(* IEC 61131-3 sources: repolevel_ST_code_completion/output/0121完整版本/repoeval_three-axis_CNC_motion/readful_result_before_fix, 5 files *)

(* ---- INIT_CNC_System.st ---- *)
FUNCTION INIT_CNC_System : BOOL
VAR_IN_OUT
	fbSMC_ReadNCFile		:	SMC_ReadNCFile;
	fbSMC_NCDecoder			:	SMC_NCDecoder;
	fbSMC_CheckVelocities	:	SMC_CheckVelocities;
	fbSMC_Interpolator		:	SMC_Interpolator;
	fbSMC_ControlAxisXByPos	:	SMC_ControlAxisByPos;
	fbSMC_ControlAxisYByPos	:	SMC_ControlAxisByPos;
	fbSMC_ControlAxisZByPos	:	SMC_ControlAxisByPos;
	fbSMC_AXISX_HOMING		:	SMC_HOMING;
	fbSMC_AXISY_HOMING		:	SMC_HOMING;
	fbSMC_AXISZ_HOMING		:	SMC_HOMING;
	fbMC_AXISX_STOP			:	MC_STOP;
	fbMC_AXISY_STOP			:	MC_STOP;
	fbMC_AXISZ_STOP			:	MC_STOP;
END_VAR
VAR_INPUT
	AxisX					:	SM3_Basic.AXIS_REF_SM3
	AxisY					:	SM3_Basic.AXIS_REF_SM3
	AxisZ					:	SM3_Basic.AXIS_REF_SM3
END_VAR
VAR
	bInitSuccess : BOOL;
END_VAR

// Reset G-code processing related function blocks
fbSMC_ReadNCFile(bExecute := FALSE);
fbSMC_NCDecoder(bExecute := FALSE, ncprog := fbSMC_ReadNCFile.ncprog);
fbSMC_CheckVelocities(bExecute := FALSE);
fbSMC_Interpolator(bExecute := FALSE);

// Stop all axes
fbMC_AXISX_STOP(Axis := AxisX, Execute := TRUE);
fbMC_AXISY_STOP(Axis := AxisY, Execute := TRUE);
fbMC_AXISZ_STOP(Axis := AxisZ, Execute := TRUE);

// Perform homing for all axes
fbSMC_AXISX_HOMING(Axis := AxisX, Execute := TRUE);
fbSMC_AXISY_HOMING(Axis := AxisY, Execute := TRUE);
fbSMC_AXISZ_HOMING(Axis := AxisZ, Execute := TRUE);

// Check if initialization was successful
bInitSuccess := fbMC_AXISX_STOP.Done AND fbMC_AXISY_STOP.Done AND fbMC_AXISZ_STOP.Done AND
                fbSMC_AXISX_HOMING.Done AND fbSMC_AXISY_HOMING.Done AND fbSMC_AXISZ_HOMING.Done;

RETURN bInitSuccess;
END_FUNCTION

(* ---- FB_TripleAxisHoming.st ---- *)
FUNCTION_BLOCK FB_TripleAxisHoming
VAR_INPUT
	bExecute			:	BOOL;				//执行回零信号
	AxisX				:	AXIS_REF;			//X轴引用
	AxisY				:	AXIS_REF;			//Y轴引用
	AxisZ				:	AXIS_REF;			//Z轴引用
	bAxisXRefSwitch		:	BOOL;				//X轴零点开关
	bAxisYRefSwitch		:	BOOL;				//Y轴零点开关
	bAxisZRefSwitch		:	BOOL;				//Z轴零点开关
	fVelocitySlow		:	REAL;				//慢速回零速度
	fVelocityFast		:	REAL;				//快速回零速度
	fAcceleration		:	REAL;				//加速度
	fDeceleration		:	REAL;				//减速度
END_VAR
VAR_OUTPUT
	bHomeOK				:	BOOL;				//三轴都回零完成
	bAxisXHomeOK		:	BOOL;				//X轴回零完成
	bAxisYHomeOK		:	BOOL;				//Y轴回零完成
	bAxisZHomeOK		:	BOOL;				//Z轴回零完成
	bBusy				:	BOOL;				//回零进行中
	bError				:	BOOL;				//错误标志
	sErrorString		:	STRING;				//错误信息字符串
END_VAR
VAR
	fbHomingX			:	SMC_HOMING;			//X轴回零功能块
	fbHomingY			:	SMC_HOMING;			//Y轴回零功能块
	fbHomingZ			:	SMC_HOMING;			//Z轴回零功能块
	bAxisXBusy			:	BOOL;				//X轴回零进行中
	bAxisYBusy			:	BOOL;				//Y轴回零进行中
	bAxisZBusy			:	BOOL;				//Z轴回零进行中
	bAxisXError			:	BOOL;				//X轴回零错误
	bAxisYError			:	BOOL;				//Y轴回零错误
	bAxisZError			:	BOOL;				//Z轴回零错误
	sAxisXErrorString	:	STRING;				//X轴错误信息
	sAxisYErrorString	:	STRING;				//Y轴错误信息
	sAxisZErrorString	:	STRING;				//Z轴错误信息
END_VAR

fbHomingX.Execute := bExecute;
fbHomingX.Axis := AxisX;
fbHomingX.ReferenceSwitch := bAxisXRefSwitch;
fbHomingX.VelocitySlow := fVelocitySlow;
fbHomingX.VelocityFast := fVelocityFast;
fbHomingX.Acceleration := fAcceleration;
fbHomingX.Deceleration := fDeceleration;

fbHomingY.Execute := bExecute;
fbHomingY.Axis := AxisY;
fbHomingY.ReferenceSwitch := bAxisYRefSwitch;
fbHomingY.VelocitySlow := fVelocitySlow;
fbHomingY.VelocityFast := fVelocityFast;
fbHomingY.Acceleration := fAcceleration;
fbHomingY.Deceleration := fDeceleration;

fbHomingZ.Execute := bExecute;
fbHomingZ.Axis := AxisZ;
fbHomingZ.ReferenceSwitch := bAxisZRefSwitch;
fbHomingZ.VelocitySlow := fVelocitySlow;
fbHomingZ.VelocityFast := fVelocityFast;
fbHomingZ.Acceleration := fAcceleration;
fbHomingZ.Deceleration := fDeceleration;

bAxisXBusy := fbHomingX.Busy;
bAxisYBusy := fbHomingY.Busy;
bAxisZBusy := fbHomingZ.Busy;

bAxisXError := fbHomingX.Error;
bAxisYError := fbHomingY.Error;
bAxisZError := fbHomingZ.Error;

sAxisXErrorString := fbHomingX.ErrorString;
sAxisYErrorString := fbHomingY.ErrorString;
sAxisZErrorString := fbHomingZ.ErrorString;

bAxisXHomeOK := fbHomingX.HomeOK;
bAxisYHomeOK := fbHomingY.HomeOK;
bAxisZHomeOK := fbHomingZ.HomeOK;

bBusy := bAxisXBusy OR bAxisYBusy OR bAxisZBusy;
bError := bAxisXError OR bAxisYError OR bAxisZError;

IF bError THEN
	IF bAxisXError THEN
		sErrorString := sAxisXErrorString;
	ELSIF bAxisYError THEN
		sErrorString := sAxisYErrorString;
	ELSIF bAxisZError THEN
		sErrorString := sAxisZErrorString;
	END_IF;
ELSE
	sErrorString := '';
END_IF;

bHomeOK := bAxisXHomeOK AND bAxisYHomeOK AND bAxisZHomeOK;
END_FUNCTION_BLOCK

(* ---- FB_TripleAxisPower.st ---- *)
FUNCTION_BLOCK FB_TripleAxisPower
VAR_INPUT
	AxisX			:	SM3_Basic.AXIS_REF_SM3			//X轴引用
	AxisY			:	SM3_Basic.AXIS_REF_SM3			//Y轴引用
	AxisZ			:	SM3_Basic.AXIS_REF_SM3			//Z轴引用
	bServoEnable	:	BOOL;				//伺服使能信号
END_VAR
VAR_OUTPUT
	bReady			:	BOOL;				//三轴都准备就绪
	bAxisXReady		:	BOOL;				//X轴准备就绪
	bAxisYReady		:	BOOL;				//Y轴准备就绪
	bAxisZReady		:	BOOL;				//Z轴准备就绪
	bError			:	BOOL;				//错误标志
	sErrorString	:	STRING;				//错误信息字符串
END_VAR
VAR
	fbPowerX		:	MC_POWER;			//X轴电源控制
	fbPowerY		:	MC_POWER;			//Y轴电源控制
	fbPowerZ		:	MC_POWER;			//Z轴电源控制
	bErrorX			:	BOOL;				//X轴错误标志
	bErrorY			:	BOOL;				//Y轴错误标志
	bErrorZ			:	BOOL;				//Z轴错误标志
END_VAR

fbPowerX(
	Enable := bServoEnable,
	bRegulatorOn := bServoEnable,
	bDriveStart := bServoEnable,
	Axis := AxisX
);
bAxisXReady := fbPowerX.Status = MC_POWER_STATUS.PoweredOn;
bErrorX := fbPowerX.Error;

fbPowerY(
	Enable := bServoEnable,
	bRegulatorOn := bServoEnable,
	bDriveStart := bServoEnable,
	Axis := AxisY
);
bAxisYReady := fbPowerY.Status = MC_POWER_STATUS.PoweredOn;
bErrorY := fbPowerY.Error;

fbPowerZ(
	Enable := bServoEnable,
	bRegulatorOn := bServoEnable,
	bDriveStart := bServoEnable,
	Axis := AxisZ
);
bAxisZReady := fbPowerZ.Status = MC_POWER_STATUS.PoweredOn;
bErrorZ := fbPowerZ.Error;

bReady := bAxisXReady AND bAxisYReady AND bAxisZReady;
bError := bErrorX OR bErrorY OR bErrorZ;

IF bError THEN
	IF bErrorX THEN
		sErrorString := 'Error in Axis X';
	ELSIF bErrorY THEN
		sErrorString := 'Error in Axis Y';
	ELSIF bErrorZ THEN
		sErrorString := 'Error in Axis Z';
	END_IF;
ELSE
	sErrorString := '';
END_IF;
END_FUNCTION_BLOCK

(* ---- FB_TripleAxisReset.st ---- *)
FUNCTION_BLOCK FB_TripleAxisReset
VAR_INPUT
	AxisX			:	SM3_Basic.AXIS_REF_SM3			//X轴引用
	AxisY			:	SM3_Basic.AXIS_REF_SM3			//Y轴引用
	AxisZ			:	SM3_Basic.AXIS_REF_SM3			//Z轴引用
	bExecute		:	BOOL;				//执行复位信号
END_VAR
VAR_OUTPUT
	bDone			:	BOOL;				//三轴都复位完成
	bBusy			:	BOOL;				//复位进行中
	bError			:	BOOL;				//错误标志
	sErrorString	:	STRING;				//错误信息字符串
END_VAR
VAR
	fbResetX		:	MC_RESET;			//X轴复位
	fbResetY		:	MC_RESET;			//Y轴复位
	fbResetZ		:	MC_RESET;			//Z轴复位
	bResetXDone		:	BOOL;				//X轴复位完成
	bResetYDone		:	BOOL;				//Y轴复位完成
	bResetZDone		:	BOOL;				//Z轴复位完成
	bResetXBusy		:	BOOL;				//X轴复位进行中
	bResetYBusy		:	BOOL;				//Y轴复位进行中
	bResetZBusy		:	BOOL;				//Z轴复位进行中
	bResetXError	:	BOOL;				//X轴复位错误
	bResetYError	:	BOOL;				//Y轴复位错误
	bResetZError	:	BOOL;				//Z轴复位错误
	sResetXErrorString	:	STRING;			//X轴错误信息
	sResetYErrorString	:	STRING;			//Y轴错误信息
	sResetZErrorString	:	STRING;			//Z轴错误信息
END_VAR

fbResetX(
	Execute := bExecute,
	Axis := AxisX
);
bResetXDone := fbResetX.Done;
bResetXBusy := fbResetX.Busy;
bResetXError := fbResetX.Error;
sResetXErrorString := fbResetX.ErrorID;

fbResetY(
	Execute := bExecute,
	Axis := AxisY
);
bResetYDone := fbResetY.Done;
bResetYBusy := fbResetY.Busy;
bResetYError := fbResetY.Error;
sResetYErrorString := fbResetY.ErrorID;

fbResetZ(
	Execute := bExecute,
	Axis := AxisZ
);
bResetZDone := fbResetZ.Done;
bResetZBusy := fbResetZ.Busy;
bResetZError := fbResetZ.Error;
sResetZErrorString := fbResetZ.ErrorID;

bDone := bResetXDone AND bResetYDone AND bResetZDone;
bBusy := bResetXBusy OR bResetYBusy OR bResetZBusy;
bError := bResetXError OR bResetYError OR bResetZError;

IF bResetXError THEN
	sErrorString := sResetXErrorString;
ELSIF bResetYError THEN
	sErrorString := sResetYErrorString;
ELSIF bResetZError THEN
	sErrorString := sResetZErrorString;
ELSE
	sErrorString := '';
END_IF;
END_FUNCTION_BLOCK

(* ---- FB_TripleAxisStop.st ---- *)
FUNCTION_BLOCK FB_TripleAxisStop
VAR_INPUT
	AxisX			:	SM3_Basic.AXIS_REF_SM3			//X轴引用
	AxisY			:	SM3_Basic.AXIS_REF_SM3			//Y轴引用
	AxisZ			:	SM3_Basic.AXIS_REF_SM3			//Z轴引用
	bExecute		:	BOOL;				//执行停止信号
	rDeceleration	:	REAL := 100.0;		//减速度
END_VAR
VAR_OUTPUT
	bDone			:	BOOL;				//三轴都停止完成
	bBusy			:	BOOL;				//停止进行中
	bError			:	BOOL;				//错误标志
	sErrorString	:	STRING;				//错误信息字符串
END_VAR
VAR
	fbStopX			:	MC_STOP;			//X轴停止
	fbStopY			:	MC_STOP;			//Y轴停止
	fbStopZ			:	MC_STOP;			//Z轴停止
	bStopXDone		:	BOOL;				//X轴停止完成
	bStopYDone		:	BOOL;				//Y轴停止完成
	bStopZDone		:	BOOL;				//Z轴停止完成
	bStopXError		:	BOOL;				//X轴停止错误
	bStopYError		:	BOOL;				//Y轴停止错误
	bStopZError		:	BOOL;				//Z轴停止错误
	sStopXErrorString:	STRING;				//X轴错误信息
	sStopYErrorString:	STRING;				//Y轴错误信息
	sStopZErrorString:	STRING;				//Z轴错误信息
END_VAR

fbStopX(
	Execute := bExecute,
	Deceleration := rDeceleration,
	Axis := AxisX
);
bStopXDone := fbStopX.Done;
bStopXError := fbStopX.Error;
sStopXErrorString := fbStopX.ErrorID;

fbStopY(
	Execute := bExecute,
	Deceleration := rDeceleration,
	Axis := AxisY
);
bStopYDone := fbStopY.Done;
bStopYError := fbStopY.Error;
sStopYErrorString := fbStopY.ErrorID;

fbStopZ(
	Execute := bExecute,
	Deceleration := rDeceleration,
	Axis := AxisZ
);
bStopZDone := fbStopZ.Done;
bStopZError := fbStopZ.Error;
sStopZErrorString := fbStopZ.ErrorID;

bDone := bStopXDone AND bStopYDone AND bStopZDone;
bBusy := fbStopX.Busy OR fbStopY.Busy OR fbStopZ.Busy;
bError := bStopXError OR bStopYError OR bStopZError;

IF bStopXError THEN
	sErrorString := CONCAT('X轴错误: ', sStopXErrorString);
ELSIF bStopYError THEN
	sErrorString := CONCAT('Y轴错误: ', sStopYErrorString);
ELSIF bStopZError THEN
	sErrorString := CONCAT('Z轴错误: ', sStopZErrorString);
ELSE
	sErrorString := '';
END_IF;
END_FUNCTION_BLOCK
